ABB RobotStudio station: Estacion_ProyectoV6_20210804-080012.rsstn

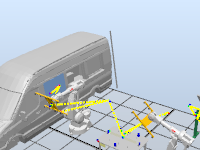
Station Estacion_ProyectoV5 (saved by RobotStudio 20.4.9280.0)
Controller ControladorBanda1, task T_ROB1: task frame (RAPID world) sits at (-1179.95, -992.74, 0) mm in the station
Controller ControladorMesa, task T_ROB1: task frame (RAPID world) sits at (-1848.82, -1848.82, 0) mm, rotated rx 0 ry 0 rz -90 deg in the station
Controller ControladorMesa
  mechanical unit ROB_1: IRB4400_60_196__03, 6 joints, base frame (-1848.82, 0, 428.3) mm
Controller ControladorBanda1
  mechanical unit ROB_1: IRB4400_60_196__03_2, 6 joints, base frame (6179.95, -657.26, 0) mm
Controller ControladorPegante
  mechanical unit ROB_1: IRB4400_60_196__03_3, 6 joints, base frame (1900, 0, 0) mm, rotated rx 0 ry 0 rz 90 deg
Controller ControladorAdhesivos
  mechanical unit ROB_1: IRB4400_60_196__03_4, 6 joints, base frame (5000, 800, 0) mm, rotated rx 0 ry 0 rz -90 deg
Layout (positions relative to the parent item):
  - Carro2 [part]
  - MesaCentrado [mechanism] at (0, 0, 0) mm; joint values [0.055, 0.055, 0.055, 0.055, 0, 0] (rad or m)
      links: L1, L2, L3, L4, L5, L6, L7
  - Vacuum Tool [mechanism] at (-1848.82, -1201.24, 2078.3) mm, rotated rx 180 ry 60 rz 90 deg
      TCP tVacuum at (0, 0, 100) mm
      links: Vacuum Tool
  - IRB4400_60_196__03 [mechanism, from Robots\IRB4400_60_196_G_03.rslib] at (-1848.82, 0, 428.3) mm, rotated rx 0 ry 0 rz -90 deg; joint values [0, 0, 0, 0, 0.5236, 0] (rad or m)
  - LogicaMesaCentrado [smart component]
      signals: DO Vidrio_Centrado, DI Pick, DI Inicio_Mesa, DI Soltar_ventana, DO Vidrio_Mesa
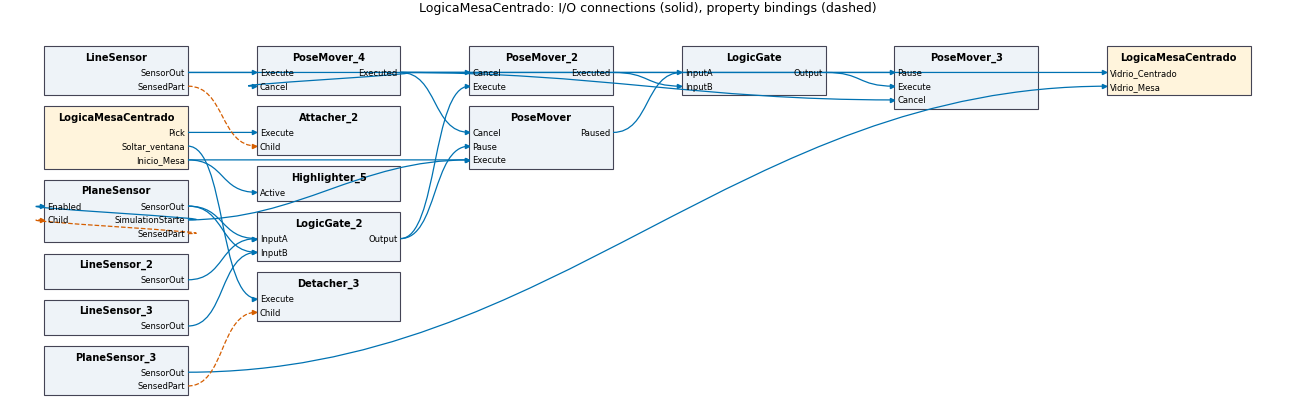
      connections:
        LineSensor.SensorOut -> PoseMover_3.Pause
        LineSensor.SensorOut -> PoseMover_4.Execute
        PoseMover.Paused -> LogicGate.InputA
        PoseMover_2.Executed -> LogicGate.InputB
        LogicGate.Output -> PoseMover_3.Execute
        PoseMover_4.Executed -> PoseMover_2.Cancel
        PoseMover_4.Executed -> PoseMover_3.Cancel
        PoseMover_4.Executed -> PoseMover.Cancel
        PoseMover_4.Executed -> PoseMover_4.Cancel
        PoseMover_4.Executed -> LogicaMesaCentrado.Vidrio_Centrado
        LogicaMesaCentrado.Pick -> Attacher_2.Execute
        LogicGate_2.Output -> PoseMover.Pause
        PlaneSensor.SensorOut -> LogicGate_2.InputA
        LogicGate_2.Output -> PoseMover_2.Execute
        PlaneSensor_2.SensorOut -> LogicGate_2.InputB
        LineSensor_2.SensorOut -> LogicGate_2.InputA
        LineSensor_3.SensorOut -> LogicGate_2.InputB
        SimulationEvents.SimulationStarted -> PhysicsControl_2.Enabled
        LogicaMesaCentrado.Soltar_ventana -> Detacher_3.Execute
        PlaneSensor_3.SensorOut -> LogicaMesaCentrado.Vidrio_Mesa
        SimulationEvents.SimulationStarted -> PoseMover.Execute
        LogicaMesaCentrado.Inicio_Mesa -> PoseMover.Execute
        LogicaMesaCentrado.Inicio_Mesa -> Highlighter_5.Active
        LineSensor.SensedPart => Attacher_2.Child
        PlaneSensor_3.SensedPart => Detacher_3.Child
        PlaneSensor_5.SensedPart => Detacher_4.Child
    - PoseMover [smart component, from Components\PoseMover.rslib]
        properties: Mechanism=MesaCentrado; Pose=2; Duration=2
    - PoseMover_2 [smart component, from Components\PoseMover.rslib]
        properties: Mechanism=MesaCentrado; Pose=1; Duration=2
    - LineSensor [smart component, from Components\LineSensor.rslib]
        properties: Start=[-0.520467 -0.0005 0.906397]; End=[-0.520467 -0.0005 0.806397]; Radius=0.003; SensedPart=(none); SensedPoint=[0 0 0]
      - _sensorPart_ [part]
    - PoseMover_3 [smart component, from Components\PoseMover.rslib]
        properties: Mechanism=MesaCentrado; Pose=3; Duration=2
    - PoseMover_4 [smart component, from Components\PoseMover.rslib]
        properties: Mechanism=MesaCentrado; Pose=1; Duration=2
    - LogicGate [smart component, from Components\LogicGate.rslib]
        properties: Operator=AND; Delay=0
    - Attacher_2 [smart component, from Components\Attacher.rslib]
        properties: Parent=Vacuum Tool; Flange=0; Child=(none); Mount=false; Offset=[0 0 0]; Orientation=[0 0 0]
    - LogicGate_2 [smart component, from Components\LogicGate.rslib]
        properties: Operator=AND; Delay=0
    - LineSensor_2 [smart component, from Components\LineSensor.rslib]
        properties: Start=[-0.37 0.383 0.906397]; End=[-0.37 0.383 0.85]; Radius=0.001; SensedPart=(none); SensedPoint=[0 0 0]
      - _sensorPart_ [part]
    - LineSensor_3 [smart component, from Components\LineSensor.rslib]
        properties: Start=[0.34 0.38 0.906397]; End=[0.34 0.38 0.85]; Radius=0.001; SensedPart=(none); SensedPoint=[0 0 0]
      - _sensorPart_ [part]
    - PlaneSensor_3 [smart component, from Components\PlaneSensor.rslib]
        properties: Origin=[-0.5 -0.0005 0.9064]; Axis1=[1 0 0]; Axis2=[0 0 -0.1]; SensedPart=(none)
      - _sensorPart_ [part]
    - Detacher_3 [smart component, from Components\Detacher.rslib]
        properties: Child=(none); KeepPosition=true
    - Highlighter_5 [smart component, from Components\Highlighter.rslib]
        properties: Object=Led_5; Color=[0 205 0]; Opacity=255
  - Ventanas [part] at (5106.38, -15819.76, 3.57) mm, rotated rx 0 ry -90 rz 89.9 deg
  - LogicaPrimeraBanda [smart component]
      signals: DO Vidrio_posicionado, DI Pick, DI Inicio, DI Repetir_ciclo
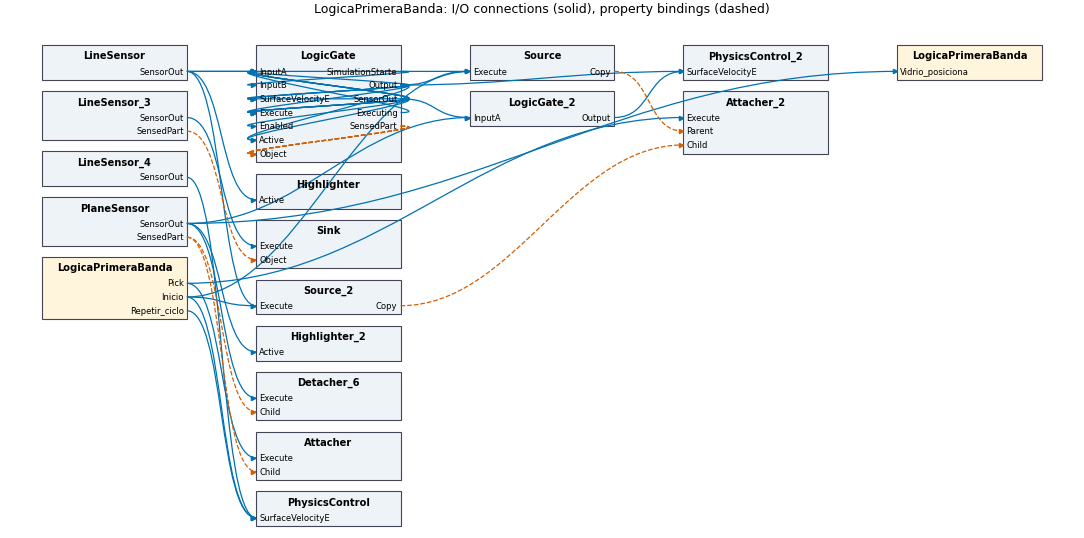
      connections:
        LineSensor.SensorOut -> LogicGate.InputA
        SimulationEvents.SimulationStarted -> LogicGate.InputB
        LogicGate.Output -> Source.Execute
        LineSensor_3.SensorOut -> Sink.Execute
        LineSensor_4.SensorOut -> LogicGate_2.InputA
        LogicGate_2.Output -> PhysicsControl.SurfaceVelocityEnabled
        LineSensor_4.SensorOut -> LinearMover2_2.Execute
        LogicGate_3.Output -> PhysicsControl.SurfaceVelocityEnabled
        LineSensor_4.SensorOut -> LogicGate_4.InputA
        LogicGate_4.Output -> LinearMover2_3.Execute
        LineSensor_4.SensorOut -> LinearMover2_3.Execute
        LineSensor_4.SensorOut -> LinearMover_2.Execute
        LineSensor_4.SensorOut -> PhysicsControl_2.Enabled
        LineSensor_4.SensorOut -> LogicGate_3.InputA
        LogicGate.Output -> PhysicsControl.SurfaceVelocityEnabled
        LineSensor_4.SensorOut -> PhysicsControl_2.SurfaceVelocityEnabled
        LineSensor_4.SensorOut -> LinearMover2.Execute
        Timer.Output -> LogicGate_2.InputA
        LogicGate_2.Output -> LineSensor_4.Active
        LinearMover2.Executing -> LogicGate.InputA
        LineSensor_4.SensorOut -> Timer.Active
        LineSensor_4.SensorOut -> PhysicsControl.SurfaceVelocityEnabled
        LineSensor_5.SensorOut -> LogicGate.InputA
        LogicGate.Output -> PhysicsControl_2.SurfaceVelocityEnabled
        LineSensor_5.SensorOut -> LogicGate_2.InputA
        LogicGate_2.Output -> PhysicsControl_2.SurfaceVelocityEnabled
        PlaneSensor.SensorOut -> LogicGate_2.InputA
        PlaneSensor.SensorOut -> LogicaPrimeraBanda.Vidrio_posicionado
        LogicaPrimeraBanda.Pick -> Attacher.Execute
        LineSensor.SensorOut -> Highlighter.Active
        PlaneSensor.SensorOut -> Highlighter_2.Active
        LogicaPrimeraBanda.Inicio -> PhysicsControl.SurfaceVelocityEnabled
        LogicaPrimeraBanda.Repetir_ciclo -> PhysicsControl.SurfaceVelocityEnabled
        PlaneSensor.SensorOut -> Detacher_6.Execute
        LogicaPrimeraBanda.Pick -> Attacher_2.Execute
        LineSensor.SensorOut -> Source.Execute
        LineSensor.SensorOut -> Source_2.Execute
        LogicaPrimeraBanda.Inicio -> Source.Execute
        LogicaPrimeraBanda.Inicio -> Source_2.Execute
        LineSensor_3.SensedPart => Sink.Object
        LineSensor_4.SensedPart => LinearMover2_3.Object
        LineSensor_4.SensedPart => LinearMover_2.Object
        LineSensor_4.SensedPart => PhysicsControl_2.Object
        LineSensor_4.SensedPart => PhysicsControl_2.Object
        PlaneSensor.SensedPart => Attacher.Child
        Source.Copy => Attacher_2.Parent
        Source_2.Copy => Attacher_2.Child
        PlaneSensor.SensedPart => Detacher_6.Child
    - LineSensor [smart component, from Components\LineSensor.rslib]
        properties: Start=[6.200046 -3.29274 1.2]; End=[7.20005 -3.29274 1.2]; Radius=0.005; SensedPart=(none); SensedPoint=[0 0 0]
      - _sensorPart_ [part]
    - Source [smart component, from Components\Source.rslib]
        properties: Source=Sostenedor; Copy=(none); Parent=(none); Position=[7.22955 -3.827103 0.706348]; Orientation=[1.5707963267949 0 -1.5707963267949]; Transient=true; PhysicsBehavior=3
    - Source_2 [smart component, from Components\Source.rslib]
        properties: Source=Ventanas; Copy=Ventanas_27; Parent=(none); Position=[6.728 -3.852702 1.112768]; Orientation=[0 -0.174532925199433 -1.5707963267949]; Transient=false; PhysicsBehavior=3
    - LineSensor_3 [smart component, from Components\LineSensor.rslib]
        properties: Start=[6.200046 -1.04274 0.75]; End=[7.200046 -1.04274 0.75]; Radius=0.005; SensedPart=(none); SensedPoint=[0 0 0]
      - _sensorPart_ [part]
    - Sink [smart component, from Components\Sink.rslib]
        properties: Object=(none)
    - SimulationEvents [smart component, from Components\SimulationEvents.rslib]
    - LineSensor_4 [smart component, from Components\LineSensor.rslib]
        properties: Start=[6.200046 -1.74274 1.2]; End=[7.200046 -1.74274 1.2]; Radius=0.001; SensedPart=(none); SensedPoint=[0 0 0]
      - _sensorPart_ [part]
    - PhysicsControl [smart component, from Components\PhysicsControl.rslib]
        properties: Object=BandaTransportadora1; Behavior=1; SurfaceVelocity=0.2
    - PhysicsControl_2 [smart component, from Components\PhysicsControl.rslib]
        properties: Object=BandaTransportadora2; Behavior=1; SurfaceVelocity=0.1
    - LogicGate_2 [smart component, from Components\LogicGate.rslib]
        properties: Operator=NOT; Delay=0
    - PlaneSensor [smart component, from Components\PlaneSensor.rslib]
        properties: Origin=[6.200046 -1.17474 1.3]; Axis1=[1 0 0]; Axis2=[0 0.2 0]; SensedPart=(none)
      - _sensorPart_ [part]
    - Attacher [smart component, from Components\Attacher.rslib]
        properties: Parent=Vacuum Tool_2; Flange=0; Child=(none); Mount=false; Offset=[0 0 0]; Orientation=[0 0 0]
    - Highlighter [smart component, from Components\Highlighter.rslib]
        properties: Object=Led_1; Color=[0 205 0]; Opacity=255
    - Highlighter_2 [smart component, from Components\Highlighter.rslib]
        properties: Object=Led_2; Color=[0 205 0]; Opacity=255
    - Attacher_2 [smart component, from Components\Attacher.rslib]
        properties: Parent=(none); Flange=0; Child=Ventanas_27; Mount=false; Offset=[0 0 0]; Orientation=[0 0 0]
    - Detacher_6 [smart component, from Components\Detacher.rslib]
        properties: Child=(none); KeepPosition=true
  - BandaTransportadora1 [part] at (6185.05, -2592.74, 600) mm, rotated rx 90 ry 0 rz -90 deg
  - BandaTransportadora2 [part] at (7236.05, -2592.74, 600) mm, rotated rx 90 ry 0 rz 90 deg
  - Vacuum Tool_2 [mechanism] at (6201.24, -1650, 1650) mm, rotated rx -180 ry 60 rz -180 deg
      TCP tVacuum at (0, 0, 100) mm
      links: Vacuum Tool
  - Sostenedor [part] at (8366.42, -15111.3, 2.34) mm, rotated rx 90 ry 0 rz -87.12 deg
  - IRB4400_60_196__03_2 [mechanism, from Robots\IRB4400_60_196_G_03.rslib] at (5000, -1650, 0) mm; joint values [0, 0, 0, 0, 0.5236, 0] (rad or m)
  - IRB4400_60_196__03_3 [mechanism, from Robots\IRB4400_60_196_G_03.rslib] at (1900, 0, 0) mm, rotated rx 0 ry 0 rz 90 deg; joint values [1.5708, -0.0873, -0.3491, 0, 1.2217, -1.5708] (rad or m)
  - Vacuum Tool_3 [mechanism] at (911.95, 0, 1901.3) mm, rotated rx -140 ry 0 rz 90 deg
      TCP tVacuum at (0, 0, 100) mm
      links: Vacuum Tool
  - BandaTransportadora2_2 [part] at (4100, -800, 600) mm, rotated rx 90 ry 0 rz 90 deg
  - BandaTransportadora1_2 [part] at (3049, -800, 600) mm, rotated rx 90 ry 0 rz -90 deg
  - IRB4400_60_196__03_4 [mechanism, from Robots\IRB4400_60_196_G_03.rslib] at (5000, 800, 0) mm, rotated rx 0 ry 0 rz -90 deg; joint values [1.5708, -0.3541, 0.1448, 0, 0.8512, 0] (rad or m)
  - Tool2 [part, from Proyecto\Tool2.rslib] at (5859.91, 800, 1418.74) mm, rotated rx -90 ry 32.93 rz 180 deg
  - LogicaSegundaBanda [smart component]
      signals: DI Poner_vidrio, DI Soltar_ventana, DI Iniciar_banda, DO Vidrio_posicionado, DI Pick
      connections:
        SimulationEvents.SimulationStarted -> Source.Execute
        LogicaSegundaBanda.Poner_vidrio -> Source.Execute
        LogicaSegundaBanda.Soltar_ventana -> Detacher.Execute
        LogicaSegundaBanda.Soltar_ventana -> Timer.Active
        PlaneSensor.SensorOut -> LogicGate_2.InputB
        LogicaSegundaBanda.Iniciar_banda -> LogicGate_2.InputA
        LogicGate_2.Output -> PhysicsControl.SurfaceVelocityEnabled
        LineSensor_2.SensorOut -> Sink.Execute
        PlaneSensor_2.SensorOut -> LogicGate_3.InputA
        LogicGate_3.Output -> PhysicsControl_2.SurfaceVelocityEnabled
        PlaneSensor_2.SensorOut -> LogicaSegundaBanda.Vidrio_posicionado
        LogicaSegundaBanda.Pick -> Attacher.Execute
        PlaneSensor_2.SensorOut -> Highlighter_3.Active
        LineSensor.SensorOut -> Highlighter_4.Active
        LineSensor.SensedPart => Detacher.Child
        LineSensor_2.SensedPart => Sink.Object
        PlaneSensor_2.SensedPart => Attacher.Child
        PlaneSensor_2.SensedPart => Detacher_2.Child
    - Source [smart component, from Components\Source.rslib]
        properties: Source=Sostenedor; Copy=(none); Parent=(none); Position=[4.094504 -1.784363 0.706348]; Orientation=[1.5707963267949 0 -1.5707963267949]; Transient=true; PhysicsBehavior=3
    - Detacher [smart component, from Components\Detacher.rslib]
        properties: Child=(none); KeepPosition=true
    - LineSensor [smart component, from Components\LineSensor.rslib]
        properties: Start=[3.09591 -1.785 1.32]; End=[4.060902 -1.785 1.32]; Radius=0.005; SensedPart=(none); SensedPoint=[0 0 0]
      - _sensorPart_ [part]
    - PhysicsControl [smart component, from Components\PhysicsControl.rslib]
        properties: Object=BandaTransportadora1_2; Behavior=1; SurfaceVelocity=0.2
    - PlaneSensor [smart component, from Components\PlaneSensor.rslib]
        properties: Origin=[3.09591 -1.4 0.71]; Axis1=[1 0 0]; Axis2=[0 1.35 0]; SensedPart=(none)
      - _sensorPart_ [part]
    - LogicGate_2 [smart component, from Components\LogicGate.rslib]
        properties: Operator=OR; Delay=0
    - LineSensor_2 [smart component, from Components\LineSensor.rslib]
        properties: Start=[3.09 0.74 0.75]; End=[4.09 0.74 0.75]; Radius=0.001; SensedPart=(none); SensedPoint=[0 0 0]
      - _sensorPart_ [part]
    - PhysicsControl_2 [smart component, from Components\PhysicsControl.rslib]
        properties: Object=BandaTransportadora2_2; Behavior=1; SurfaceVelocity=0.1
    - PlaneSensor_2 [smart component, from Components\PlaneSensor.rslib]
        properties: Origin=[3.09 0.52002 1.3]; Axis1=[1 0 0]; Axis2=[0 0.2 0]; SensedPart=(none)
      - _sensorPart_ [part]
    - Sink [smart component, from Components\Sink.rslib]
        properties: Object=(none)
    - LogicGate_3 [smart component, from Components\LogicGate.rslib]
        properties: Operator=NOT; Delay=0
    - Attacher [smart component, from Components\Attacher.rslib]
        properties: Parent=Vacuum Tool_3; Flange=0; Child=(none); Mount=false; Offset=[0 0 0]; Orientation=[0 0 0]
    - Highlighter_3 [smart component, from Components\Highlighter.rslib]
        properties: Object=Led_4; Color=[0 205 0]; Opacity=255
    - Highlighter_4 [smart component, from Components\Highlighter.rslib]
        properties: Object=Led_3; Color=[0 205 0]; Opacity=255
  - AplicadorPegante [mechanism] at (0, 0, 0) mm; joint values [0] (rad or m)
      links: L1, L2
  - Carro [part] at (-2500.01, -3277.23, 0) mm
  - LogicaVidrioCarro [smart component]
      signals: DI Ventana_carro
      connections:
        LogicaVidrioCarro.Ventana_carro -> Detacher_5.Execute
        PlaneSensor_6.SensorOut -> Attacher.Execute
        PlaneSensor_6.SensedPart => Detacher_5.Child
        PlaneSensor_6.SensedPart => Attacher.Child
    - PlaneSensor_6 [smart component, from Components\PlaneSensor.rslib]
        properties: Origin=[-2.905 0.106665 1.72757]; Axis1=[-0.1 0 0]; Axis2=[0 0.1 0]; SensedPart=Ventanas_21
      - _sensorPart_ [part]
    - Detacher_5 [smart component, from Components\Detacher.rslib]
        properties: Child=Ventanas_21; KeepPosition=true
    - Attacher [smart component, from Components\Attacher.rslib]
        properties: Parent=Carro; Flange=0; Child=Ventanas_21; Mount=false; Offset=[0 0 0]; Orientation=[0 0 0]
  - Tablero_1 [part] at (7216.05, -3882.74, 520) mm
  - Led_1 [part] at (7236.05, -3832.74, 470) mm
  - Tablero_2 [part] at (7236.05, -1302.74, 520) mm, rotated rx 0 ry 0 rz 180 deg
  - Led_2 [part] at (7236.05, -1452.74, 470) mm
  - Led_4 [part] at (4100, 340, 470) mm
  - Tablero_4 [part] at (4100, 490, 520) mm, rotated rx 0 ry 0 rz 180 deg
  - Led_3 [part] at (4100, -2040, 470) mm
  - Tablero_3 [part] at (4080, -2090, 520) mm
  - Tablero_5 [part] at (-553.01, -465, 701.4) mm, rotated rx 0 ry 0 rz -90 deg
  - Led_5 [part] at (-503.01, -485, 651.4) mm, rotated rx 0 ry 0 rz -90 deg
  - Ventanas_21 [part] at (-2906.1, 117.57, 1735.84) mm, rotated rx -179.95 ry -7 rz 0 deg
  - Ventanas_23 [part] at (6733.85, -2280.11, 1063.86) mm, rotated rx 0 ry -22.64 rz -90.76 deg
  - Ventanas_25 [part] at (6737.22, -2814.43, 1062.09) mm, rotated rx 0 ry -23.32 rz -90.88 deg
  - Ventanas_27 [part] at (6724.3, -3356.45, 1109.28) mm, rotated rx 0 ry -14.37 rz -90.01 deg
Attachment: Vacuum Tool_2 is attached to IRB4400_60_196__03_2 / Link6
Attachment: Vacuum Tool_3 is attached to IRB4400_60_196__03_3 / Link6
Attachment: Tool2 is attached to IRB4400_60_196__03_4 / Link6
Attachment: Vacuum Tool is attached to IRB4400_60_196__03 / Link6
Attachment: LogicaPrimeraBanda is attached to Led_4
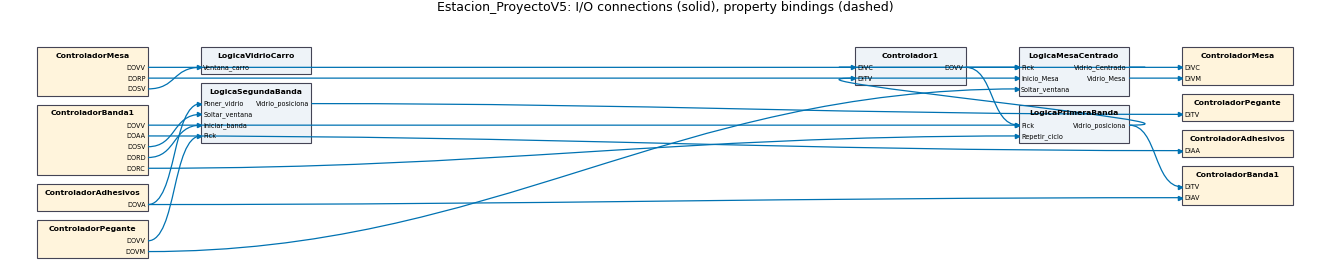
Station logic (signal -> signal, property => property):
  LogicaMesaCentrado.Vidrio_Centrado -> Controlador1.DIVC
  Controlador1.DOVV -> LogicaMesaCentrado.Pick
  LogicaMesaCentrado.Vidrio_Centrado -> ControladorMesa.DIVC
  ControladorMesa.DOVV -> LogicaMesaCentrado.Pick
  ControladorMesa.DORP -> LogicaMesaCentrado.Inicio_Mesa
  LogicaPrimeraBanda.Vidrio_posicionado -> ControladorBanda1.DITV
  ControladorBanda1.DOVV -> LogicaPrimeraBanda.Pick
  LogicaPrimeraBanda.Vidrio_posicionado -> ControladorBanda1.DITV
  ControladorBanda1.DOVV -> LogicaPrimeraBanda.Pick
  ControladorBanda1.DOAA -> ControladorAdhesivos.DIAA
  ControladorAdhesivos.DOVA -> ControladorBanda1.DIAV
  ControladorAdhesivos.DOVA -> LogicaSegundaBanda.Poner_vidrio
  ControladorBanda1.DOSV -> LogicaSegundaBanda.Soltar_ventana
  ControladorBanda1.DORD -> LogicaSegundaBanda.Iniciar_banda
  LogicaSegundaBanda.Vidrio_posicionado -> ControladorPegante.DITV
  ControladorPegante.DOVV -> LogicaSegundaBanda.Pick
  ControladorPegante.DOVM -> LogicaMesaCentrado.Soltar_ventana
  LogicaMesaCentrado.Vidrio_Mesa -> ControladorMesa.DIVM
  ControladorMesa.DOSV -> LogicaVidrioCarro.Ventana_carro
  ControladorBanda1.DORC -> LogicaPrimeraBanda.Repetir_ciclo
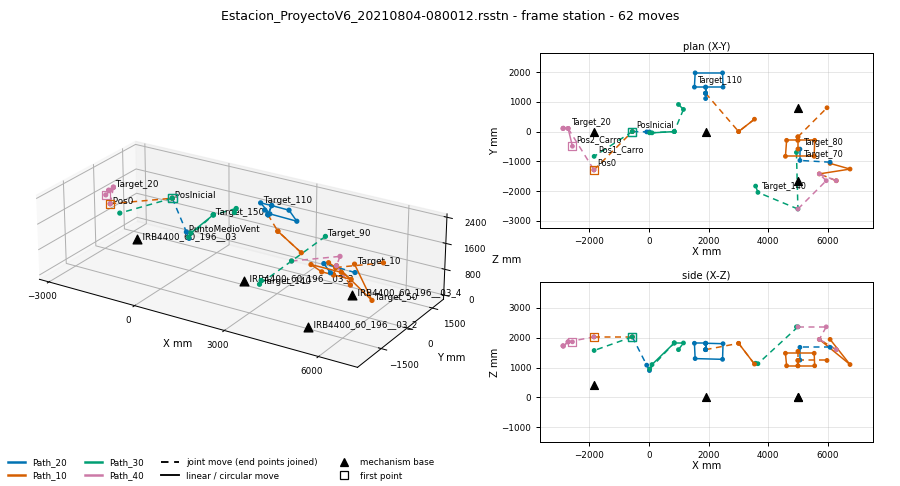
[picture p0: tool path of Estacion_ProyectoV6_20210804-080012.rsstn in frame station, 62 of 62 moves have a stored position in this frame; points joined in program order, loops and branches not executed]
Targets, tools, work objects and paths stored in the station, written as RAPID:
! task (no controller)
MODULE CalibData
  TASK PERS wobjdata Workobject_1:=[FALSE,TRUE,"",[[-622.5,-535,771.397],[1,0,0,0]],[[0,0,0],[1,0,0,0]]];
  TASK PERS tooldata Tooldata_1:=[TRUE,[[0,0,0],[1,0,0,0]],[1,[0,0,1],[1,0,0,0],0,0,0]];
ENDMODULE

! task T_ROB1
MODULE CalibData
  PERS tooldata tVacuum:=[TRUE,[[0,0,100],[1,0,0,0]],[18,[0,0,66.666666667],[1,0,0,0],0,0,0]];
  TASK PERS wobjdata Workobject_1:=[FALSE,TRUE,"",[[-1313.815,1226.315,771.397],[0.707106781,0,0,0.707106781]],[[0,0,0],[1,0,0,0]]];
ENDMODULE

! task T_ROB1
MODULE Module1
  CONST robtarget Pos0:=[[-1226.315,-752.846096908,1256.9],[0.353553391,0.612372436,0.612372436,-0.353553391],[0,0,0,0],[9E+09,9E+09,9E+09,9E+09,9E+09,9E+09]];
  CONST robtarget TomarVentana:=[[636.85,523,127.153],[0,0.707106781,0.707106781,0],[0,0,0,0],[9E+09,9E+09,9E+09,9E+09,9E+09,9E+09]];
  CONST robtarget PuntoMedio1:=[[267.497993061,270.074268995,351.133526228],[0.073258901,0.703302172,0.703299637,-0.073272162],[0,-1,1,0],[9E+09,9E+09,9E+09,9E+09,9E+09,9E+09]];
  CONST robtarget PosInicial:=[[61.531096908,535,1256.9],[0.5,0,0.866025404,0],[1,0,-1,0],[9E+09,9E+09,9E+09,9E+09,9E+09,9E+09]];
  CONST robtarget PuntoMedioVent:=[[544.537164154,524.921391442,308.422917653],[0.092194571,0.619720217,0.779388872,-0.000009273],[1,-1,0,0],[9E+09,9E+09,9E+09,9E+09,9E+09,9E+09]];
  CONST robtarget Pos1_Carro:=[[-1220.780000251,-297.409948892,800.672994623],[0.500000009,0.499999986,-0.499999991,0.500000014],[0,0,1,0],[9E+09,9E+09,9E+09,9E+09,9E+09,9E+09]];
  CONST robtarget Pos2_Carro:=[[-1949.609936804,42.660022246,1091.332977127],[0.707032595,0.192887484,-0.680289946,-0.010242956],[-1,0,1,0],[9E+09,9E+09,9E+09,9E+09,9E+09,9E+09]];
  CONST robtarget VentanaCarro:=[[-2251.761031846,651.449110404,944.881043321],[0.707106845,-0.000000687,-0.707106717,0.000000199],[-2,1,0,0],[9E+09,9E+09,9E+09,9E+09,9E+09,9E+09]];
  CONST robtarget Target_10:=[[-2094.835519591,640.954336723,1091.333033624],[0.65822494,-0.058788633,-0.704658699,-0.25834075],[-1,0,1,0],[9E+09,9E+09,9E+09,9E+09,9E+09,9E+09]];
  CONST robtarget Target_20:=[[-2094.835494649,640.954150658,1091.332999686],[0.684311147,0.025566154,-0.706644482,-0.178096049],[-2,0,1,0],[9E+09,9E+09,9E+09,9E+09,9E+09,9E+09]];
  CONST robtarget Target_30:=[[-2094.839990026,640.949981815,1091.332992071],[0.707106781,-0.000000009,-0.707106781,0.000000018],[-2,-1,2,0],[9E+09,9E+09,9E+09,9E+09,9E+09,9E+09]];
  CONST robtarget Target_40:=[[-2256.141,649.346,946.665],[0.662620048,0,-0.748955721,0],[-2,-1,2,0],[9E+09,9E+09,9E+09,9E+09,9E+09,9E+09]];
  CONST robtarget Target_50:=[[-2292.100031529,649.346107297,946.665025888],[0.707106781,-0.000000159,-0.707106781,0.000000151],[-2,-1,2,0],[9E+09,9E+09,9E+09,9E+09,9E+09,9E+09]];
  CONST robtarget Target_60:=[[-2289.285027332,650.682570667,946.665005738],[0.707106774,-0.000000128,-0.707106788,0.000000147],[-2,-1,2,0],[9E+09,9E+09,9E+09,9E+09,9E+09,9E+09]];
  CONST robtarget Target_70:=[[-2289.285017532,646.861310529,959.920954139],[0.707106777,-0.000000126,-0.707106785,0.000000123],[-2,-1,2,0],[9E+09,9E+09,9E+09,9E+09,9E+09,9E+09]];
  CONST robtarget Target_80:=[[-2289.285023772,646.534994264,949.174029414],[0.707106789,-0.000000116,-0.707106773,0.000000117],[-2,-1,2,0],[9E+09,9E+09,9E+09,9E+09,9E+09,9E+09]];
  CONST robtarget Target_90:=[[-2289.285015286,643.630043899,948.639011289],[0.707106785,-0.000000198,-0.707106777,0.000000167],[-2,-1,2,0],[9E+09,9E+09,9E+09,9E+09,9E+09,9E+09]];
  CONST robtarget Target_100:=[[-2267.5,638.905,958.357],[0.662620048,0,-0.748955721,0],[-2,-1,2,0],[9E+09,9E+09,9E+09,9E+09,9E+09,9E+09]];
  PROC Path_20()
    MoveJ PosInicial,v500,z50,tVacuum\WObj:=Workobject_1;
    MoveJ PuntoMedioVent,v500,z10,tVacuum\WObj:=Workobject_1;
    MoveL TomarVentana,v150,fine,tVacuum\WObj:=Workobject_1;
    SetDO DOVV,1;
    WaitTime 1;
    SetDO DOVV,0;
  ENDPROC
  PROC main()
    SetDO DORP,0;
    SetDO DOVV,0;
    SetDO DOSV,0;
    WaitDI DIVM,1;
    Path_10;
    WaitDI DIVC,1;
    Path_20;
    Path_30;
    WaitTime 2;
    Path_40;
  ENDPROC
  PROC Path_10()
    MoveJ Pos0,v500,z50,tVacuum\WObj:=Workobject_1;
    MoveJ PosInicial,v500,z20,tVacuum\WObj:=Workobject_1;
    SetDO DORP,1;
    WaitTime 1;
    SetDO DORP,0;
  ENDPROC
  PROC Path_30()
    MoveJ PosInicial,v500,z200,tVacuum\WObj:=Workobject_1;
    MoveJ Pos1_Carro,v500,z200,tVacuum\WObj:=Workobject_1;
  ENDPROC
  PROC Path_40()
    MoveJ Pos2_Carro,v500,z50,tVacuum\WObj:=Workobject_1;
    MoveL Target_20,v200,fine,tVacuum\WObj:=Workobject_1;
    MoveL Target_30,v200,fine,tVacuum\WObj:=Workobject_1;
    MoveL Target_40,v100,fine,tVacuum\WObj:=Workobject_1;
    MoveL Target_100,v100,fine,tVacuum\WObj:=Workobject_1;
    SetDO DOSV,1;
    WaitTime 1;
    SetDO DOSV,0;
    MoveL Target_100,v100,fine,tVacuum\WObj:=Workobject_1;
    MoveL Target_40,v100,fine,tVacuum\WObj:=Workobject_1;
    MoveL Target_30,v200,fine,tVacuum\WObj:=Workobject_1;
    MoveJ Pos0,v500,z50,tVacuum\WObj:=Workobject_1;
  ENDPROC
ENDMODULE

! task T_ROB1
MODULE CalibData
  TASK PERS wobjdata Workobject_1:=[FALSE,TRUE,"",[[7372.5,-100.002,695],[0.707106781,0,0,-0.707106781]],[[0,0,0],[1,0,0,0]]];
  PERS tooldata tVacuum:=[TRUE,[[0,0,100],[1,0,0,0]],[18,[0,0,66.666666667],[1,0,0,0],0,0,0]];
ENDMODULE

! task T_ROB1
MODULE Module1
  CONST robtarget Pos0:=[[557.262,95.3,905],[0.353553391,-0.612372436,0.612372436,0.353553391],[0,0,0,0],[9E+09,9E+09,9E+09,9E+09,9E+09,9E+09]];
  CONST robtarget Target_10:=[[-23.865,-111.711,1249.666],[0.001231355,-0.803814383,0.000977914,0.59487811],[0,0,-1,0],[9E+09,9E+09,9E+09,9E+09,9E+09,9E+09]];
  CONST robtarget Target_20:=[[327.749,-473.857,1249.666],[0.148845925,-0.789910592,-0.10446398,0.585639329],[-1,0,-1,0],[9E+09,9E+09,9E+09,9E+09,9E+09,9E+09]];
  CONST robtarget Target_50:=[[166.289,557.454,405],[0.001884056,-0.803868748,-0.002628602,0.59479793],[0,0,-2,0],[9E+09,9E+09,9E+09,9E+09,9E+09,9E+09]];
  CONST robtarget Target_60:=[[-64.547,-111.711,983.332],[0.000822342,-0.554379087,0.001331591,0.832262806],[0,1,-2,0],[9E+09,9E+09,9E+09,9E+09,9E+09,9E+09]];
  CONST robtarget Target_70:=[[-123.908,-1125.343,983.332],[0.000392562,-0.282508617,0.001514665,0.959263485],[0,1,-2,0],[9E+09,9E+09,9E+09,9E+09,9E+09,9E+09]];
  CONST robtarget Target_80:=[[-504.424,-1125.343,555],[0.000455398,-0.324734343,0.001496011,0.945803976],[0,1,-2,0],[9E+09,9E+09,9E+09,9E+09,9E+09,9E+09]];
  CONST robtarget Target_90:=[[-391.677844574,-1242.277711435,1671.141056565],[0.051702006,0.168382035,-0.000019411,-0.984364969],[1,2,-2,0],[9E+09,9E+09,9E+09,9E+09,9E+09,9E+09]];
  CONST robtarget Target_100:=[[1507.500114911,-1192.546013658,1671.141056565],[0.985381053,0.004427133,0.168323826,0.025916618],[-2,2,-2,0],[9E+09,9E+09,9E+09,9E+09,9E+09,9E+09]];
  CONST robtarget Target_120:=[[737.282,-2613.085,447.979],[0.638077524,0.002155819,-0.769969107,-0.000030075],[-2,-1,-1,0],[9E+09,9E+09,9E+09,9E+09,9E+09,9E+09]];
  CONST robtarget Target_130:=[[557.260013658,-242.305859524,1671.141042042],[0.678443712,-0.11589251,0.122153452,0.715095511],[0,2,-2,0],[9E+09,9E+09,9E+09,9E+09,9E+09,9E+09]];
  CONST robtarget Target_140:=[[949.005949401,-2535.272894899,433.049039714],[0.439744571,0.102523926,-0.891201443,-0.043284458],[-2,-1,-1,0],[9E+09,9E+09,9E+09,9E+09,9E+09,9E+09]];
  PROC Path_10()
    MoveJ Pos0,v2500,z10,tVacuum\WObj:=Workobject_1;
    MoveJ Target_20,v2500,z10,tVacuum\WObj:=Workobject_1;
    MoveL Target_50,v600,fine,tVacuum\WObj:=Workobject_1;
    SetDO DOVV,1;
    WaitTime 1;
    SetDO DOVV,0;
    MoveL Target_10,v1000,fine,tVacuum\WObj:=Workobject_1;
  ENDPROC
  PROC main()
    SetDO DOVV,0;
    SetDO DOAA,0;
    SetDO DOSV,0;
    SetDO DORD,0;
    WaitDI DITV,1;
    Path_10;
    Path_20;
    WaitDI DIAV,1;
    Path_30;
    WaitTime 1;
    Path_40;
  ENDPROC
  PROC Path_20()
    MoveJ Target_60,v2500,z10,tVacuum\WObj:=Workobject_1;
    MoveJ Target_70,v2500,z10,tVacuum\WObj:=Workobject_1;
    MoveL Target_80,v600,fine,tVacuum\WObj:=Workobject_1;
    SetDO DOAA,1;
    WaitTime 1;
    SetDO DOAA,0;
  ENDPROC
  PROC Path_30()
    MoveJ Target_90,v2500,z10,tVacuum\WObj:=Workobject_1;
    MoveJ Target_100,v3000,z10,tVacuum\WObj:=Workobject_1;
    MoveJ Target_140,v600,z10,tVacuum\WObj:=Workobject_1;
    MoveL Target_120,v200,fine,tVacuum\WObj:=Workobject_1;
    SetDO DOSV,1;
    WaitTime 1;
    SetDO DOSV,0;
  ENDPROC
  PROC Path_40()
    MoveJ Target_100,v3000,z50,tVacuum\WObj:=Workobject_1;
    SetDO DORD,1;
    MoveJ Target_130,v3000,z50,tVacuum\WObj:=Workobject_1;
    MoveJ Target_20,v3000,z50,tVacuum\WObj:=Workobject_1;
    MoveJ Pos0,v3000,fine,tVacuum\WObj:=Workobject_1;
    SetDO DORD,0;
  ENDPROC
ENDMODULE

! task T_ROB1
MODULE CalibData
  PERS tooldata tVacuum:=[TRUE,[[0,0,100],[1,0,0,0]],[18,[0,0,66.666666667],[1,0,0,0],0,0,0]];
  TASK PERS wobjdata Workobject_1:=[FALSE,TRUE,"",[[3056.5,700,695],[0.707106781,0,0,-0.707106781]],[[0,0,0],[1,0,0,0]]];
ENDMODULE

! task T_ROB1
MODULE Module1
  CONST robtarget Target_10:=[[-587.846096908,-1156.5,905],[0,0.866025404,0,-0.5],[0,0,0,0],[9E+09,9E+09,9E+09,9E+09,9E+09,9E+09]];
  CONST robtarget Target_20:=[[284.276,484.084,420.823],[0.583124412,-0.006706358,-0.81234092,-0.004814039],[-1,0,0,0],[9E+09,9E+09,9E+09,9E+09,9E+09,9E+09]];
  CONST robtarget Target_30:=[[700,-48.000032362,1117.070073277],[0.048300167,-0.159891842,0.943828808,0.285112036],[-2,-1,0,0],[9E+09,9E+09,9E+09,9E+09,9E+09,9E+09]];
  CONST robtarget Target_40:=[[-408.499975009,-1156.499987803,1117.070075287],[0.167451245,0.780448334,-0.554327201,-0.235757996],[0,-1,0,0],[9E+09,9E+09,9E+09,9E+09,9E+09,9E+09]];
  CONST robtarget Target_50:=[[-587.846096908,-1156.5,905],[0,0.866025404,0,-0.5],[0,0,0,0],[9E+09,9E+09,9E+09,9E+09,9E+09,9E+09]];
  CONST robtarget Target_60:=[[-587.818,-1156.5,905.032],[0,-0.382683432,0,0.923879533],[-1,0,0,0],[9E+09,9E+09,9E+09,9E+09,9E+09,9E+09]];
  CONST robtarget Target_70:=[[-792.678987422,-1156.5,1120.093056966],[0,-0.382683362,0,0.923879562],[0,0,0,0],[9E+09,9E+09,9E+09,9E+09,9E+09,9E+09]];
  CONST robtarget Target_80:=[[-792.679,-571.342,1105.093],[0,-0.382683432,0,0.923879533],[-1,-1,0,0],[9E+09,9E+09,9E+09,9E+09,9E+09,9E+09]];
  CONST robtarget Target_90:=[[-1271.774,-587.233,580.067],[0,-0.382683432,0,0.923879533],[-1,-1,0,0],[9E+09,9E+09,9E+09,9E+09,9E+09,9E+09]];
  CONST robtarget Target_100:=[[-1271.774,-1507.798,605.067],[0,-0.382683432,0,0.923879533],[0,0,-1,0],[9E+09,9E+09,9E+09,9E+09,9E+09,9E+09]];
  CONST robtarget Target_110:=[[-792.679,-1532.013,1120.093],[0,-0.382683432,0,0.923879533],[0,0,-1,0],[9E+09,9E+09,9E+09,9E+09,9E+09,9E+09]];
  CONST robtarget Target_120:=[[-210.625568644,-2067.125568644,905.0330734],[0.353553381,0.353553445,0.146446632,-0.853553368],[0,0,0,0],[9E+09,9E+09,9E+09,9E+09,9E+09,9E+09]];
  CONST robtarget Target_130:=[[-44.107502257,-1900.607446078,1129.69420725],[0.130885423,0.868162816,0.359604763,-0.315985355],[0,-1,-1,0],[9E+09,9E+09,9E+09,9E+09,9E+09,9E+09]];
  CONST robtarget Target_140:=[[700,-2208.826881831,1129.69420725],[0.241844714,0.664463059,0.66446302,-0.241844728],[1,0,-1,0],[9E+09,9E+09,9E+09,9E+09,9E+09,9E+09]];
  CONST robtarget Target_150:=[[700,-2208.826902693,1129.694224755],[0.00000001,0.000000028,0.939692623,-0.342020138],[1,-1,-1,0],[9E+09,9E+09,9E+09,9E+09,9E+09,9E+09]];
  CONST robtarget Target_160:=[[742.162,-3035.55,252.034],[0,0,1,0],[1,-1,-1,0],[9E+09,9E+09,9E+09,9E+09,9E+09,9E+09]];
  CONST robtarget Target_170:=[[742.162027464,-2956.77498855,405.146051096],[0.000000019,0.000000016,1,-0.000000002],[1,0,-1,0],[9E+09,9E+09,9E+09,9E+09,9E+09,9E+09]];
  CONST robtarget Target_180:=[[742.162007854,-2986.89293643,385.423977652],[-0.000000068,0.000000016,1,-0.000000018],[1,-1,-1,0],[9E+09,9E+09,9E+09,9E+09,9E+09,9E+09]];
  PROC Path_10()
    MoveJ Target_10,v3000,z50,tVacuum\WObj:=Workobject_1;
    MoveJ Target_30,v3000,z50,tVacuum\WObj:=Workobject_1;
    MoveL Target_20,v500,fine,tVacuum\WObj:=Workobject_1;
    SetDO DOVV,1;
    WaitTime 1;
    SetDO DOVV,0;
    MoveJ Target_30,v3000,z50,tVacuum\WObj:=Workobject_1;
  ENDPROC
  PROC main()
    SetDO DOVV,0;
    SetDO DOVM,0;
    WaitDI DITV,1;
    Path_10;
    Path_20;
    Path_30;
  ENDPROC
  PROC Path_20()
    MoveJ Target_40,v2000,z10,tVacuum\WObj:=Workobject_1;
    MoveJ Target_50,v2000,z10,tVacuum\WObj:=Workobject_1;
    MoveJ Target_60,v2000,z10,tVacuum\WObj:=Workobject_1;
    MoveL Target_70,v500,fine,tVacuum\WObj:=Workobject_1;
    MoveL Target_80,v500,fine,tVacuum\WObj:=Workobject_1;
    MoveL Target_90,v500,fine,tVacuum\WObj:=Workobject_1;
    MoveL Target_100,v500,fine,tVacuum\WObj:=Workobject_1;
    MoveL Target_110,v500,fine,tVacuum\WObj:=Workobject_1;
    MoveL Target_70,v500,fine,tVacuum\WObj:=Workobject_1;
    MoveJ Target_60,v2000,z10,tVacuum\WObj:=Workobject_1;
  ENDPROC
  PROC Path_30()
    MoveJ Target_120,v2000,z10,tVacuum\WObj:=Workobject_1;
    MoveJ Target_130,v2000,z10,tVacuum\WObj:=Workobject_1;
    MoveJ Target_140,v2000,z10,tVacuum\WObj:=Workobject_1;
    MoveJ Target_150,v2000,z10,tVacuum\WObj:=Workobject_1;
    MoveL Target_170,v500,fine,tVacuum\WObj:=Workobject_1;
    MoveL Target_160,v500,fine,tVacuum\WObj:=Workobject_1;
    SetDO DOVM,1;
    WaitTime 1;
    SetDO DOVM,0;
    MoveJ Target_150,v2000,z10,tVacuum\WObj:=Workobject_1;
  ENDPROC
ENDMODULE

! task T_ROB1
MODULE CalibData
  TASK PERS wobjdata Workobject_1:=[FALSE,TRUE,"",[[5549.625000325,-907.85240122,1476.986869221],[0.669107891,-0.22856355,0.230678247,0.668461577]],[[0,0,0],[1,0,0,0]]];
  TASK PERS tooldata Adhesivo:=[TRUE,[[0,0,215],[1,0,0,0]],[1,[0,0,1],[1,0,0,0],0,0,0]];
ENDMODULE

! task T_ROB1
MODULE Module1
  CONST robtarget Target_10:=[[723.549036654,550.359957719,258.991982571],[0.00156353,0.999060335,0.000014401,0.043312849],[-1,0,-1,0],[9E+09,9E+09,9E+09,9E+09,9E+09,9E+09]];
  CONST robtarget Target_20:=[[742.157990906,549.688540162,44.799865386],[0.00156353,0.999060335,0.000014401,0.043312849],[-1,0,-1,0],[9E+09,9E+09,9E+09,9E+09,9E+09,9E+09]];
  CONST robtarget Target_30:=[[742.098019093,-12.540710712,46.557047594],[0.00156353,0.999060335,0.000014401,0.043312849],[0,-1,0,0],[9E+09,9E+09,9E+09,9E+09,9E+09,9E+09]];
  CONST robtarget Target_40:=[[59.432963171,3.265733321,48.972332058],[0.00156353,0.999060335,0.000014401,0.043312849],[0,-1,0,0],[9E+09,9E+09,9E+09,9E+09,9E+09,9E+09]];
  CONST robtarget Target_50:=[[59.535954151,968.795012183,45.954682465],[0.00156353,0.999060335,0.000014401,0.043312849],[-1,0,-1,0],[9E+09,9E+09,9E+09,9E+09,9E+09,9E+09]];
  CONST robtarget Target_60:=[[742.198497629,929.434683321,43.613012932],[0.00156353,0.999060335,0.000014401,0.043312849],[-1,0,-1,0],[9E+09,9E+09,9E+09,9E+09,9E+09,9E+09]];
  CONST robtarget Pos0:=[[212.653026713,550.376340944,246.79732732],[0.001523489,0.981457168,-0.000351873,-0.191675203],[0,0,0,0],[9E+09,9E+09,9E+09,9E+09,9E+09,9E+09]];
  CONST robtarget Target_70:=[[1494.235839934,-424.644219336,862.061499137],[0.410883805,0.7058329,0.576274293,0.029704459],[1,-1,0,0],[9E+09,9E+09,9E+09,9E+09,9E+09,9E+09]];
  PROC Path_10()
    MoveJ Pos0,v2000,z10,Adhesivo\WObj:=Workobject_1;
    MoveJ Target_10,v1500,z10,Adhesivo\WObj:=Workobject_1;
    MoveL Target_20,v800,fine,Adhesivo\WObj:=Workobject_1;
    MoveL Target_30,v800,fine,Adhesivo\WObj:=Workobject_1;
    MoveL Target_40,v800,fine,Adhesivo\WObj:=Workobject_1;
    MoveL Target_50,v800,fine,Adhesivo\WObj:=Workobject_1;
    MoveL Target_60,v800,fine,Adhesivo\WObj:=Workobject_1;
    MoveL Target_20,v800,fine,Adhesivo\WObj:=Workobject_1;
    MoveJ Target_10,v1500,z10,Adhesivo\WObj:=Workobject_1;
    MoveJ Target_70,v3000,z10,Adhesivo\WObj:=Workobject_1;
    SetDO DOVA,1;
    WaitTime 1;
    SetDO DOVA,0;
  ENDPROC
  PROC main()
    SetDO DOVA,0;
    WaitDI DIAA,1;
    Path_10;
  ENDPROC
ENDMODULE

